{attribute 'qualified_only'}
VAR_GLOBAL CONSTANT
	iAOChannelCount : INT := 50;
	
END_VAR
VAR_GLOBAL
	in_cmd								: ARRAY [1..iAOChannelCount] OF REAL;
	fdbk								: ARRAY [1..iAOChannelCount] OF REAL;
	iAO							AT %Q*	: ARRAY [1..iAOChannelCount] OF INT;
	ifdbk							AT %I*	: ARRAY [1..iAOChannelCount] OF INT;
END_VAR

(* stored: Version 1.1.0.1, ProductVersion 3.1.4024.12
   GVL GVL_AnalogOutputs: Id {563f42e0-5daa-4bb3-9ff0-cdc92f4f2c6f} *)
